// Mitsubishi GX Works2 project: analogInput   PLC: FX3G

// global labels: Global1
VAR_GLOBAL
  aI_TempOut AT D14 : INT;  (* AI_0 Датчик наружней температуры D8030 *)
  aI_TempSupply AT D15 : INT;  (* AI_1 Датчик притока (температуры подачи в помещение)  D8031 *)
  xInit AT M15 : BOOL;
  xUserStart AT M11 : BOOL;  (* Переменная изменяемая Пользователем для разрешения работы *)
  xAlarm AT M0 : BOOL;
  iStep AT D50 : INT;
END_VAR

// task Task_01 (event TRUE, interval 0, priority 31): POU_01

PROGRAM POU_01
IF xInit =  FALSE THEN  iStep := 0 ; ELSE iStep := 10;  END_IF;
	R23941 := 3;
	CASE iStep OF
	0:
	MOV(TRUE,  1, R23940);
	xInit := TRUE;
	iStep := 10;
	10:
	;
	
	END_CASE;
END_PROGRAM
